{attribute 'GeneratedUsingTerminal: AMP8000-0030-0103-0103'}
{attribute addProperty BoxType "AMP8000-0030-0103-0103"}
{attribute addProperty Id "Power_supply_controlwordAT %Q*UINT2"}
{attribute addProperty CRC "1695495302"}
{attribute addProperty Size "2"}
TYPE DeviceMain_Outputs_650F3486 EXTENDS OutputBase_10CEE7DE :
STRUCT
	{attribute addProperty Name "Power_supply_controlword"}
	Power_supply_controlword AT %Q* : UINT;
END_STRUCT
END_TYPE

(* stored: Version 1.2.0.0, ProductVersion 3.1.4024.9
   DUT DeviceMain_Outputs_650F3486: Id {3a67af41-f28e-4e74-a77f-7d7ec714bbd4} *)
